(* IEC 61131-3 sources: AXOpen/src/integrations/app/src/Examples, 1 file *)

(* ---- VMTest.st ---- *)
NAMESPACE VmT
    {S7.extern=ReadWrite}
    CLASS VmTest
        VAR PUBLIC
            {#ix-set:AttributeName = "My integer"}
            my_int : INT;
            {#ix-set:AttributeName = "My string"}
            my_string : STRING;
            {#ix-set:AttributeName = "My bool"}
            my_bool : BOOL;
        END_VAR
    END_CLASS
END_NAMESPACE
